# EPICS SNL sequencer program: siteApps/globalInterlock-1-1/ginterlockApp/src/sncTBxGInt.stt
program sncTBxGInt
option +r;
option +c;
option -a;

%%#include <math.h>

float Etc_setpt[6];
assign Etc_setpt to {
	"SCL31-CDL01:EBx01-CV7501:Setpt",		"IF-CDL07:EBx01-CV7501:Setpt",
	"SCL31-CDL01:EBx01-CV7401:Setpt",		"SCL31-CDL01:EBx01-CV7402:Setpt",
	"IF-CDL07:EBx01-CV7401:Setpt",			"IF-CDL07:EBx01-CV7402:Setpt"
};

int Etc_setmanuclose[2];
assign Etc_setmanuclose to {
	"SCL32-CDL02:VBx01-XV7301:SetManuClose","SCL22-CDL06:VBx25-XV7301:SetManuClose"
};

int etc_intstat[8];
assign etc_intstat to {
	"SCL31-CDL01:EBx01-CV7501:IntStatTBxPT7506G", "IF-CDL07:EBx01-CV7501:IntStatTBxPT7546G",
	"SCL31-CDL01:EBx01-CV7401:IntStatTBxPT7303G", "SCL31-CDL01:EBx01-CV7402:IntStatTBxPT7303G",
	"IF-CDL07:EBx01-CV7401:IntStatTBxPT7343G",	  "IF-CDL07:EBx01-CV7402:IntStatTBxPT7343G"
	"SCL32-CDL02:VBx01-XV7301:IntStatTBxPT7203G", "SCL22-CDL06:VBx25-XV7301:IntStatTBxPT7243G"
};

monitor etc_intstat;
evflag  evETCIntstat;
sync etc_intstat  evETCIntstat;

float Tbx_setpt[4];
assign Tbx_setpt to {
	"Cryo-CDL000:TBx01-CV7504:Setpt", "Cryo-CDL00:TBx01-CV7545:Setpt",
	"Cryo-CDL000:TBx01-CV7304:Setpt", "Cryo-CDL00:TBx01-CV7344:Setpt"
};

int tbx_intstat[4];
assign tbx_intstat to {
	"Cryo-CDL000:TBx01-CV7504:IntStatPT7506G", "Cryo-CDL00:TBx01-CV7545:IntStatPT7546G",
	"Cryo-CDL000:TBx01-CV7304:IntStatPT7303G", "Cryo-CDL00:TBx01-CV7344:IntStatPT7343G"
};
monitor tbx_intstat;
evflag  evTBXIntstat;
sync tbx_intstat  evTBXIntstat;

int idxcount = 8;
ss ssTBxInterlock {
	state init {
		when(TRUE)
		{

		}state TBxGInterlock
	}

	state TBxGInterlock
	{
		when(efTest(evETCIntstat))
		{
			int i = 0;
			for( ; i < idxcount;i++)
			{
				if (i < 6 && etc_intstat[i] == 1) {
					Etc_setpt[i] = 0;
					pvPut(Etc_setpt[i], SYNC);
				} else {
					//Shut-off valve close
					Etc_setmanuclose[i] = 1;
					pvPut(Etc_setmanuclose[i], SYNC);
				};
			}
			efClear(evETCIntstat);
		} state Step1
	}

	state Step1
	{
		when(efTest(evTBXIntstat))
		{
			int i = 0;
			for( ; i < 4;i++)
			{
				if (tbx_intstat[i] == 1) {
					Tbx_setpt[i] = 0;
					pvPut(Tbx_setpt[i], SYNC);
				} ;
			};
			efClear(evTBXIntstat);
		} state GoDelay
	}

	state GoDelay
	{
		when(delay(1.0))
		{
			efSet(evETCIntstat);
			efSet(evTBXIntstat);
		}state TBxGInterlock
	}
}
